{attribute 'linkalways'} 
{attribute 'no_explicit_call' := 'This FB is a CLASS and must be accessed using methods or properties'}
{attribute 'enable_dynamic_creation'}
FUNCTION_BLOCK PUBLIC SyslogClient
VAR
	// Properties
	_hostname : STRING := '127.0.0.1';
	_port : UINT := 514;
	app_name : STRING(32) := 'TwinCAT_PLC';
    
	// Internal Logic
	socket_handle : Tc2_TcpIp.T_HSocket;
	socket_create : Tc2_TcpIp.Fb_SocketUdpCreate;
	udp_send : Tc2_TcpIp.Fb_SocketUdpSendTo;
    
    log_payload : STRING(512);
    timestamp : STRING(32);
    get_time : Tc2_Utilities.NT_GetTime;
    
    state : INT := 0;
END_VAR

PROPERTY PUBLIC AppName : STRING(255)
GET // PUBLIC
AppName := app_name;
END_GET
SET // PUBLIC
app_name := AppName;
END_SET
END_PROPERTY

METHOD PUBLIC Execute
CASE state OF
    0: // Idle
        
    10: // Fetch Timestamp
        get_time(START := TRUE);
        IF NOT get_time.BUSY AND NOT get_time.ERR THEN
            UpdateTimestamp();
            get_time(START := FALSE);
            state := 20;
        ELSIF get_time.ERR THEN
            get_time(START := FALSE);
            state := 0;
        END_IF

    20: // Maintain Socket
        IF socket_handle.handle = 0 THEN
			socket_create(
				bExecute := TRUE,
				sLocalHost := _hostname,
				nLocalPort := 4444
			);
			IF NOT socket_create.bBusy AND NOT socket_create.bError THEN
				socket_handle := socket_create.hSocket;
				socket_create(bExecute := FALSE);
			END_IF
		ELSE
			state := 30;
		END_IF

    30: // Dispatch UDP
        udp_send(
            hSocket := socket_handle, 
            sRemoteHost := _hostname, 
            nRemotePort := _port,
            pSrc := ADR(log_payload), 
            cbLen := INT_TO_UDINT(Tc2_Standard.Len(log_payload)), 
            bExecute := TRUE
		);
            
        IF NOT udp_send.bBusy AND NOT udp_send.bError THEN
            udp_send(bExecute := FALSE);
            state := 0; 
        END_IF
END_CASE
END_METHOD

//FB_Init is always available implicitly and it is used primarily for initialization.
//The return value is not evaluated. For a specific influence, you can also declare the
//methods explicitly and provide additional code there with the standard initialization
//code. You can evaluate the return value.
METHOD FB_Init: BOOL
VAR_INPUT
    bInitRetains: BOOL; // TRUE: the retain variables are initialized (reset warm / reset cold)
    bInCopyCode: BOOL;  // TRUE: the instance will be copied to the copy code afterward (online change)
	hostname : STRING(15);
	port : UINT;   
END_VAR
THIS^._hostname := hostname;
THIS^._port := port;
END_METHOD

PROPERTY PUBLIC Hostname : STRING(15)
GET // PUBLIC
Hostname := _hostname;
END_GET
SET // PUBLIC
_hostname := Hostname;
ResetConnection();
END_SET
END_PROPERTY

METHOD PUBLIC LogCustomFormat : BOOL
VAR_INPUT
    data : Tc2_System.T_MaxString;
END_VAR
SendLog(6, data);
LogCustomFormat := TRUE;
END_METHOD

METHOD PUBLIC LogStandardFormat : BOOL
VAR_INPUT
    data : Tc2_System.T_MaxString;
    instance_path : Tc2_System.T_MaxString;
    log_level: Nepionic_Log.LogLevel;
END_VAR
VAR
    empty_attrs : ARRAY[0..9] OF Nepionic_Log.LogAttribute;
END_VAR
LogStandardFormat := LogWithAttributes(data, instance_path, log_level, empty_attrs, 0);
END_METHOD

/// LogCore stub. Structured attributes are not represented in RFC 5424 structured data
/// by this backend — attrs/attr_count are silently ignored and the message is sent as-is.
METHOD PUBLIC LogWithAttributes : BOOL
VAR_INPUT
    data : Tc2_System.T_MaxString;
    instance_path : Tc2_System.T_MaxString;
    log_level : Nepionic_Log.LogLevel;
    attrs : ARRAY[0..9] OF Nepionic_Log.LogAttribute;
    attr_count : USINT;
END_VAR
VAR
    syslog_severity : INT;
END_VAR
CASE log_level OF
    Nepionic_Log.LogLevel.Debug:       syslog_severity := 7;
    Nepionic_Log.LogLevel.Information: syslog_severity := 6;
    Nepionic_Log.LogLevel.Warning:     syslog_severity := 4;
    Nepionic_Log.LogLevel.Error:       syslog_severity := 3;
    Nepionic_Log.LogLevel.Fatal:       syslog_severity := 2;
ELSE
    syslog_severity := 6;
END_CASE

SendLog(syslog_severity, data);
LogWithAttributes := TRUE;
END_METHOD

PROPERTY PUBLIC Port : UINT
GET // PUBLIC
Port := _port;
END_GET
SET // PUBLIC
_port := Port;
ResetConnection();
END_SET
END_PROPERTY

METHOD PRIVATE ResetConnection
END_METHOD

METHOD PUBLIC SendLog
VAR_INPUT
	severity : INT; // 0: Emerg ... 7: Debug
	message  : STRING(255);
END_VAR
VAR_INST
	priority : INT;
END_VAR
// Facility 1 (User) * 8 + severity
priority := 8 + severity;

// Build RFC 5424 String: <PRI>1 TIMESTAMP HOSTNAME APPNAME - - - MESSAGE
log_payload := Tc2_System.Concat('<', INT_TO_STRING(priority));
log_payload := Tc2_System.Concat(log_payload, '>1 ');
log_payload := Tc2_System.Concat(log_payload, timestamp);
log_payload := Tc2_System.Concat(log_payload, ' ');
log_payload := Tc2_System.Concat(log_payload, hostname);
log_payload := Tc2_System.Concat(log_payload, ' ');
log_payload := Tc2_System.Concat(log_payload, app_name);
log_payload := Tc2_System.Concat(log_payload, ' - - - ');
log_payload := Tc2_System.Concat(log_payload, message);

state := 10;
END_METHOD

METHOD PRIVATE UpdateTimestamp
timestamp := WORD_TO_STRING(get_time.TimeStr.wYear);
timestamp := Tc2_System.Concat(timestamp, '-');
timestamp := Tc2_System.Concat(timestamp, Tc2_System.Right(Tc2_System.Concat('0', WORD_TO_STRING(get_time.TimeStr.wMonth)), 2));
timestamp := Tc2_System.Concat(timestamp, '-');
timestamp := Tc2_System.Concat(timestamp, Tc2_System.Right(Tc2_System.Concat('0', WORD_TO_STRING(get_time.TimeStr.wDay)), 2));
timestamp := Tc2_System.Concat(timestamp, 'T');
timestamp := Tc2_System.Concat(timestamp, Tc2_System.Right(Tc2_System.Concat('0', WORD_TO_STRING(get_time.TimeStr.wHour)), 2));
timestamp := Tc2_System.Concat(timestamp, ':');
timestamp := Tc2_System.Concat(timestamp, Tc2_System.Right(Tc2_System.Concat('0', WORD_TO_STRING(get_time.TimeStr.wMinute)), 2));
timestamp := Tc2_System.Concat(timestamp, ':');
timestamp := Tc2_System.Concat(timestamp, Tc2_System.Right(Tc2_System.Concat('0', WORD_TO_STRING(get_time.TimeStr.wSecond)), 2));
timestamp := Tc2_System.Concat(timestamp, 'Z');
END_METHOD

END_FUNCTION_BLOCK

(* stored: Version 1.1.0.1
   POU SyslogClient: Id {65da91dd-37c6-440b-88b6-2bbd59c30aea}, SpecialFunc None
   Property AppName: Id {69b1bab1-fea0-43a1-afbb-318bd2a15499}
   Get Get: Id {d1a68ea8-4c25-44c9-8464-0ab7d31af665}
   Set Set: Id {56f39b8b-17d5-4370-8706-3e2eb12efdd8}
   Method Execute: Id {195b89c6-f1f5-4050-85b6-8f519ff13b66}
   Method FB_Init: Id {0eb4f292-1f79-4499-b771-0df51136a6b7}
   Property Hostname: Id {63a46136-b9b3-4aa1-83f2-16cc510dd4ef}
   Get Get: Id {f957e786-f414-464f-9932-caf59f193812}
   Set Set: Id {06c4f3ac-0956-4cf9-ae24-b9d9161b0031}
   Method LogCustomFormat: Id {f0d8d91e-6caf-4eae-a169-50c736d993ec}
   Method LogStandardFormat: Id {9140b159-05a9-4388-b4b0-63120e6cfb32}
   Method LogWithAttributes: Id {d7a2971c-4c99-41e1-85ea-60a86360624e}
   Property Port: Id {53f57cd8-5a6f-43d4-8e65-106edc432c72}
   Get Get: Id {8e619826-137d-4410-984e-d6317a0c67c7}
   Set Set: Id {01812b08-4913-4a95-b63f-a7d7a22a697a}
   Method ResetConnection: Id {b64eb69f-6a8c-4d88-8067-e37badc0a559}
   Method SendLog: Id {ecac61fe-f83a-437b-8841-ec7e55496033}
   Method UpdateTimestamp: Id {1139199d-f0fc-4772-ae4f-78d53bfd33e7} *)
